{attribute addProperty BoxType "EP3356-0022-0016"}
{attribute addProperty Id "RMB_StatusAT %I*RMB_Status_7F71BA301620RMB_Value_INT32AT %I*RMB_Value_INT_1F5759573240RMB_ControlAT %Q*RMB_Control_D468E5481620WcStateAT %I*WcState_98A4DF7520.250InfoDataAT %I*InfoData_BC63D37F80100"}
{attribute addProperty CRC "2862345699"}
{attribute addProperty SizeInBites "146"}
{attribute addProperty SizeInBytes "18.25"}
TYPE EP3356_AAE78EE2 :
STRUCT
	{attribute addProperty Name "RMB_Status"}
	RMB_Status : RMB_Status_7F71BA30;
	{attribute addProperty Name "RMB_Value_INT32"}
	RMB_Value_INT32 : RMB_Value_INT_1F575957;
	{attribute addProperty Name "RMB_Control"}
	RMB_Control : RMB_Control_D468E548;
	{attribute addProperty Name "WcState"}
	WcState : WcState_98A4DF75;
	{attribute addProperty Name "InfoData"}
	InfoData : InfoData_BC63D37F;
END_STRUCT
END_TYPE

(* stored: Version 1.2.0.0, ProductVersion 3.1.4024.9
   DUT EP3356_AAE78EE2: Id {60c85f72-b447-42b8-909d-50b1af16c01a} *)
